TYPE ST_PrioFunctions :
STRUCT
	PickupFunctionNumber	: E_FunctionNumber;
	DepositFunctionNumber	: E_FunctionNumber;
	HighestPriority			: BOOL;
END_STRUCT
END_TYPE

(* stored: Version 1.1.0.1, ProductVersion 3.1.4022.12
   DUT ST_PrioFunctions: Id {0aaa9978-0e12-4597-98fb-d8270d3aad2c} *)
